FUNCTION_BLOCK IA_FPTO (* ISOBUS Adapter for Front Power Take off (FPTO) *)
  (* Standard: ISO 11783-7; Classification: PGN 65092; Description: Copyright (c) 2024-2026 HR Agrartechnik GmbH This program and the accompanying materials are made available under the terms of the Eclipse Public License 2.0 which is available at https://www.eclipse.org/legal/epl-2.0/ SPDX-License-Identifier: EPL-2.0 *)
  (* Version 1.2, 2026-09-17, Franz Höpfinger, HR Agrartechnik GmbH, Bugfix (Franz: 'IA_VDS hat einen Bug, moeglicherweise alle anderen auch'): .IND->TIMEOUT.E1 ergaenzt (analog IA_VDS) - bisher wurde TIMEOUT.E1 NUR von .TIMEOUT gefeuert (Timeout-Beginn), nie beim Eintreffen einer normalen Botschaft (.IND) - TIMEOUT.D1 (Q_timeout=FALSE) wurde also gesetzt, aber nie an den TIMEOUT-Plug propagiert, sobald der Timeout wieder endete. *)
  (* Version 1.1, 2026-09-16, Franz Höpfinger, HR Agrartechnik GmbH, E_D_FF_ANY-Aenderungsfilter fuer SPEED/SPEED_SET ergaenzt (analog IA_RPTO v1.1). *)
  PACKAGE isobus::tecu;
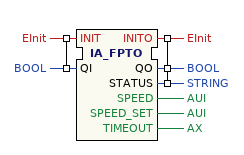
  EVENT_INPUT
    INIT : EInit WITH QI; (* Service Initialization *)
  END_EVENT
  EVENT_OUTPUT
    INITO : EInit WITH QO, STATUS; (* Initialization Confirm *)
  END_EVENT
  VAR_INPUT
    QI : BOOL; (* Event Input Qualifier *)
  END_VAR
  VAR_OUTPUT
    QO : BOOL; (* Event Output Qualifier *)
    STATUS : STRING;
  END_VAR
  PLUGS
    SPEED : adapter::types::unidirectional::AUI; (* Front PTO output shaft speed *)
    SPEED_SET : adapter::types::unidirectional::AUI; (* Front PTO output shaft speed set point *)
    TIMEOUT : adapter::types::unidirectional::AX; (* Timeout Status *)
  END_PLUGS
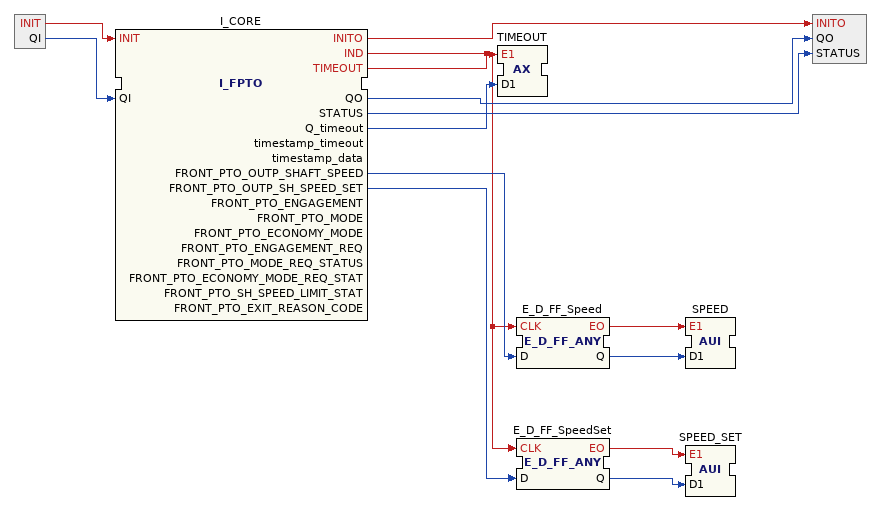
  FBS
    I_CORE : isobus::tecu::I_FPTO;
    E_D_FF_Speed : iec61499::events::E_D_FF_ANY;
    E_D_FF_SpeedSet : iec61499::events::E_D_FF_ANY;
  END_FBS
  EVENT_CONNECTIONS
    INIT TO I_CORE.INIT;
    I_CORE.INITO TO INITO;
    I_CORE.IND TO E_D_FF_Speed.CLK;
    E_D_FF_Speed.EO TO SPEED.E1;
    I_CORE.IND TO E_D_FF_SpeedSet.CLK;
    E_D_FF_SpeedSet.EO TO SPEED_SET.E1;
    I_CORE.TIMEOUT TO TIMEOUT.E1;
    I_CORE.IND TO TIMEOUT.E1;
  END_CONNECTIONS
  DATA_CONNECTIONS
    QI TO I_CORE.QI;
    I_CORE.QO TO QO;
    I_CORE.STATUS TO STATUS;
    I_CORE.FRONT_PTO_OUTP_SHAFT_SPEED TO E_D_FF_Speed.D;
    E_D_FF_Speed.Q TO SPEED.D1;
    I_CORE.FRONT_PTO_OUTP_SH_SPEED_SET TO E_D_FF_SpeedSet.D;
    E_D_FF_SpeedSet.Q TO SPEED_SET.D1;
    I_CORE.Q_timeout TO TIMEOUT.D1;
  END_CONNECTIONS
END_FUNCTION_BLOCK
